(* IEC 61131-3 sources: plc_on_fpga_riscv_hybrid/RV_FPGA_PLC_IDE_Projects/PWM_Test_2, 1 file *)

(* ---- PWM_Test_2.il ---- *)
VAR
    PWM_1   : PWM
    PWM_2   : PWM
END_VAR

PROGRAM PWM_Test_2
    R1 :
        CAL PWM_1(
            F  := 2,
            DC := 25,
            Q  => %LEDG.0)
        CAL PWM_2(
            F  := 2,
            DC := 50,
            Q  => %LEDG.1)
END_PROGRAM
